//Progress
IF eTMCFile_Int = eSelectTMCFile.eDontUseTMCFile THEN 
	IF bBusyInt THEN byProgress := (REAL_TO_BYTE(F_Scalvalue(x:= UDINT_TO_REAL(udiCounterSymbol), x1:= 0, y1:= 0, x2:= UDINT_TO_REAL(stSymbolUploadInfo.udiSymbols), y2:= 100)) + byProgressClearVarInterface + byProgressCopyArray) / 3; END_IF 	
ELSE
	IF bBusyInt THEN byProgress := (REAL_TO_BYTE(F_Scalvalue(x:= UDINT_TO_REAL(udiCounterSymbol), x1:= 0, y1:= 0, x2:= UDINT_TO_REAL(stSymbolUploadInfo.udiSymbols), y2:= 100)) + byProgressClearVarInterface + byProgressParseDocument + byProgressSubItems + byProgressCopyArray) / 5; END_IF 
END_IF

END_FUNCTION_BLOCK

(* stored: Version 1.1.0.1, ProductVersion 3.1.4024.12
   POU FB_VarInfo_V3: Id {8df5b901-c557-4fea-8acc-951ef8db7ab8}, SpecialFunc None *)
